(* PLC project test_st_in_main_and_nested_sfc.project, CODESYS CODESYS V3.5 SP14 Patch 1 *)
(* stored: creationDateTime 2019-02-25T12:02:33.1733892, modificationDateTime 2019-02-25T11:52:31.5665239 *)

PROGRAM PLC_PRG
  VAR
    i : INT := 0;
    j : INT := 0;
    k : INT := 0;
  END_VAR

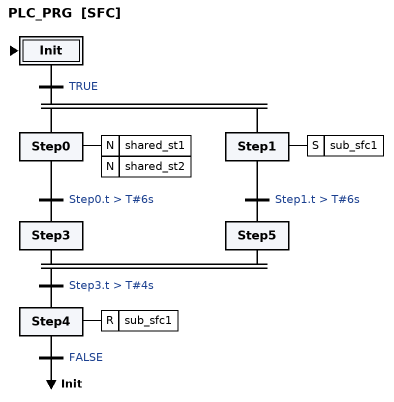
INITIAL_STEP Init:
END_STEP
TRANSITION FROM Init TO (Step0, Step1)
  := TRUE;
END_TRANSITION
STEP Step0:
  shared_st1(N);
  shared_st2(N);
END_STEP
TRANSITION FROM Step0 TO Step3
  := Step0.t > T#6s;
END_TRANSITION
STEP Step3:
END_STEP
TRANSITION FROM (Step3, Step5) TO Step4
  := Step3.t > T#4s;
END_TRANSITION
STEP Step1:
  sub_sfc1(S);
END_STEP
TRANSITION FROM Step1 TO Step5
  := Step1.t > T#6s;
END_TRANSITION
STEP Step5:
END_STEP
STEP Step4:
  sub_sfc1(R);
END_STEP
TRANSITION FROM Step4 TO Init
  := FALSE;
END_TRANSITION

ACTION sub_sfc1:
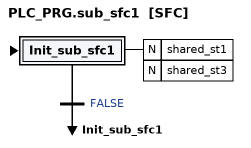
INITIAL_STEP Init_sub_sfc1:
  shared_st1(N);
  shared_st3(N);
END_STEP
TRANSITION FROM Init_sub_sfc1 TO Init_sub_sfc1
  := FALSE;
END_TRANSITION
END_ACTION

ACTION shared_st1:
                i := i + 1;
              
END_ACTION

ACTION shared_st2:
                j := j + 1;
              
END_ACTION

ACTION shared_st3:
                k := k + 1;
              
END_ACTION
END_PROGRAM
